TYPE ST_PneumaticAxisControl :
STRUCT
    bStartExtend AT %Q*: BOOL; //Move cylinder to Extend
    bStartRetract AT %Q*: BOOL; //Move cylinder to Retract

END_STRUCT
END_TYPE

(* stored: Version 1.1.0.1, ProductVersion 3.1.4024.5
   DUT ST_PneumaticAxisControl: Id {60247fff-ef28-4c35-9aa0-027d94fb1099} *)
